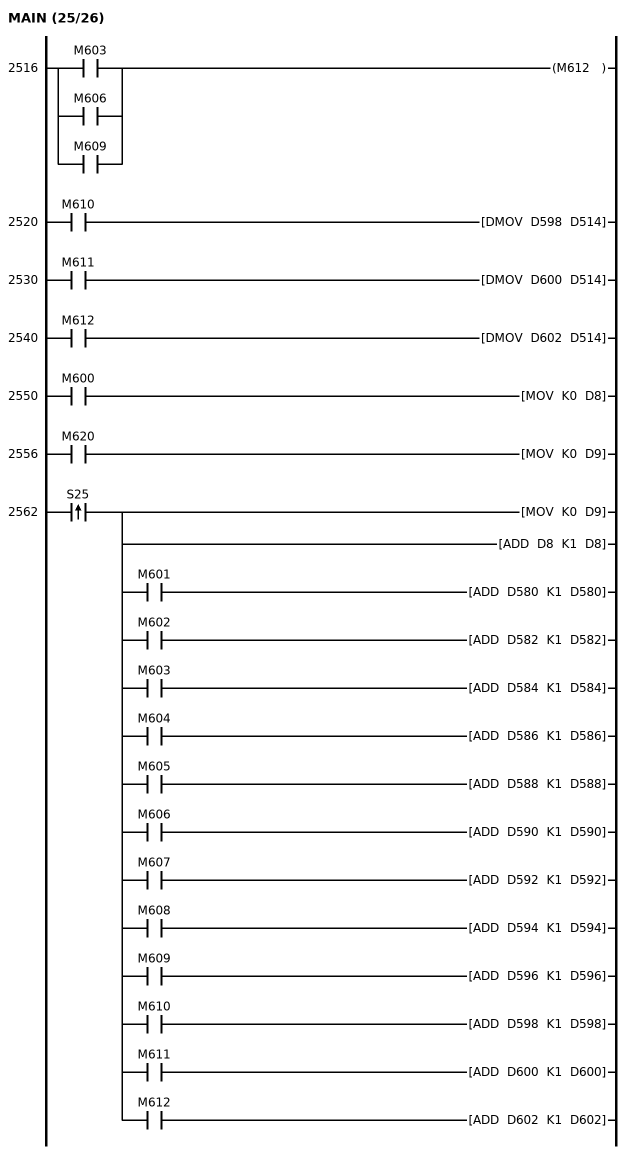
[picture p24: ladder of MAIN, rungs at steps 2516 to 2562]
2516  LD      M603
      OR      M606
      OR      M609
      OUT     M612
2520  LD      M610
      DMOV    D598 D514
2530  LD      M611
      DMOV    D600 D514
2540  LD      M612
      DMOV    D602 D514
2550  LD      M600
      MOV     K0 D8
2556  LD      M620
      MOV     K0 D9
2562  LDP     S25
      MOV     K0 D9
      ADD     D8 K1 D8
      MPS
      AND     M601
      ADD     D580 K1 D580
      MRD
      AND     M602
      ADD     D582 K1 D582
      MRD
      AND     M603
      ADD     D584 K1 D584
      MRD
      AND     M604
      ADD     D586 K1 D586
      MRD
      AND     M605
      ADD     D588 K1 D588
      MRD
      AND     M606
      ADD     D590 K1 D590
      MRD
      AND     M607
      ADD     D592 K1 D592
      MRD
      AND     M608
      ADD     D594 K1 D594
      MRD
      AND     M609
      ADD     D596 K1 D596
      MRD
      AND     M610
      ADD     D598 K1 D598
      MRD
      AND     M611
      ADD     D600 K1 D600
      MPP
      AND     M612
      ADD     D602 K1 D602
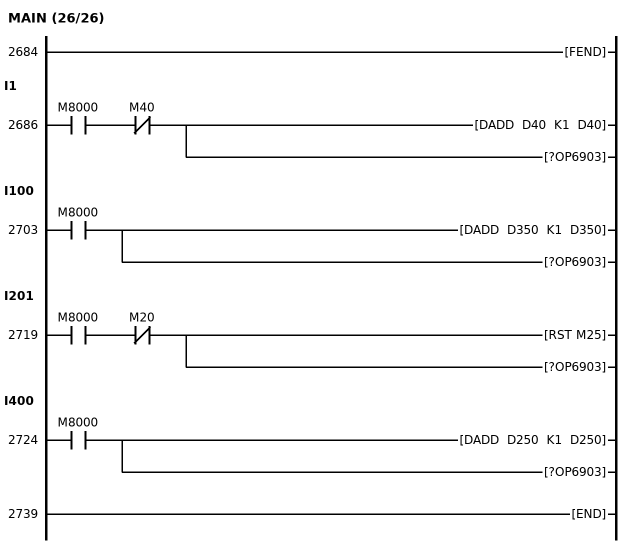
2684  FEND
      I1
2686  LD      M8000
      ANI     M40
      DADD    D40 K1 D40
      ?OP6903
      I100
2703  LD      M8000
      DADD    D350 K1 D350
      ?OP6903
      I201
2719  LD      M8000
      ANI     M20
      RST     M25
      ?OP6903
      I400
2724  LD      M8000
      DADD    D250 K1 D250
      ?OP6903
2739  END
END_PROGRAM
